// TIA Portal V16 export
// export: Created 2024-09-05T17:40:14.8581069Z, ExportSetting WithDefaults, DisplayName Totally Integrated Automation Portal, DisplayVersion V16 Update 6, DisplayName TIA Portal Version Control Interface, DisplayVersion V16 Update 2, DisplayName TIA Portal Openness, DisplayVersion V16 Update 6, DisplayName STEP 7 Professional, DisplayVersion V16 Update 6, DisplayName STEP 7 Safety, DisplayVersion V16, DisplayName WinCC Advanced, DisplayVersion V16 Update 6
TYPE "UDT_ProductionReadings"
// stored: IsFailsafeCompliant false
   STRUCT
      Enable : Bool;   // Reading active
      ReaderNumber : USInt;   // Fix (1 to 5) or Manual (10)
      "Name" : WString[30];   // Name of Label to read
      LabelType : USInt;   // Master NFP, 2nd NFP, Component Label, batch label
      ReferenceToFound : WString[30];   // Reference to be found
      ReferenceStartPosition : USInt;   // Position of reference to be found
      ReferenceLenght : USInt;   // Reference Lenght
      MasterReadingNumber : USInt;   // Reading number of master NFP
      LinkedMasterNumber : USInt;   // Linked number to master NFP
      Message : Array[1..6] of "UDT_IJCoreReadingMessage";   // IJCore Message
   END_STRUCT;
END_TYPE
